(* CODESYS project Tc3_Mc3PlanarMotion.library
   TcLibraryId: Beckhoff Automation GmbH|Tc3_Mc3PlanarMotion|3.4.67.0
   Company: Beckhoff Automation GmbH
   DefaultNamespace: Tc3_Mc3PlanarMotion
   Version: 3.4.67.0
   Placeholder: Tc3_Mc3PlanarMotion
   Title: Tc3_Mc3PlanarMotion

Project tree, tasks and I/O mapping:
  libraries: Tc3_Physics, 3.4.67.0 (Beckhoff Automation GmbH)
  Version/
    global variables Global_Version
  POUs/
    function block MC_PlanarEnvironment [ST]: FB_init, FB_reinit, FB_exit, Clear, AddStator, CreateBoundary, Update, AddToGroup, RemoveFromGroup, GetPlanarObjectInfo
    function block MC_PlanarPart [ST]: FB_init, FB_reinit, FB_exit, Initialize, ActivatePosition, ForceEnable, AllowEnable, ForceDisable, Reset, GetPosition, IsInitialized, State, IsDisableForced, PositionIndex
    function block MC_PlanarGroup [ST]: FB_init, FB_reinit, FB_exit, Enable, Disable, Reset, Update
    function block MC_PlanarTrack [ST]: FB_init, FB_reinit, FB_exit, Clear, AppendPosition, AppendLine, AppendCircle, CloseLoop, StartFromTrack, EndAtTrack, StartFromTrackAdvanced, EndAtTrackAdvanced, Enable, Disable, Reset, GetArcLengthClosestTo, GetPositionAt, GetLength, GetPlanarObjectInfo, Update, AddToGroup, RemoveFromGroup
    function block MC_PlanarTrackTrail [ST]: FB_init, FB_reinit, FB_exit, Clear, AddTrack, GetTrackOidAt, TrackCount
    function block MC_PlanarMover [ST]: FB_init, FB_reinit, FB_exit, MoveToPosition, JoinTrack, LeaveTrack, MoveOnTrack, GearInPosOnTrack, GearInPosOnTrackWithMasterMover, MoveX, MoveY, MoveZ, MoveA, MoveB, MoveC, MoveRelativeX, MoveRelativeY, MoveRelativeC, MoveVelocityX, MoveVelocityY, MoveVelocityC, AdoptTrackOrientation, Halt, Enable, Disable, Reset, Update, SetPosition, StartExternalSetpointGeneration, StopExternalSetpointGeneration, SetExternalSetpoint, SetExternalSetpointReferenceId, RaiseError, AddToGroup, RemoveFromGroup, GetPositionOnCurrentPart, GetTrackTrailInformation, GetPlanarObjectInfo, MoverHardwareOid
    function block MC_PlanarFeedbackBase [ST]: FB_init, FB_reinit, FB_exit
    function block MC_PlanarFeedback [ST]: FB_init, FB_reinit, FB_exit, Update
    function block MC_PlanarFeedbackInSync [ST]: FB_init, FB_reinit, FB_exit
    function block MC_PlanarFeedbackGearInPosOnTrack [ST]: FB_init, FB_reinit, FB_exit, Update
    function block MC_PlanarFeedbackGearInPosOnTrackWithMasterMover [ST]: FB_init, FB_reinit, FB_exit, Update
  DUTs/
    Enums/
      data type MC_SET_POSITION_MODE
      data type MC_DIRECTION
      data type MC_SYNC_DIRECTIONS
      data type EPlanarObjectType
    Structs/
      data type PlanarObjectInfo
      data type ST_MoveToPositionOptions
      data type ST_JoinTrackOptions
      data type ST_LeaveTrackOptions
      data type ST_MoveOnTrackOptions
      data type ST_GearInPosOnTrackOptions
      data type ST_GearInPosOnTrackWithMasterMoverOptions
      data type ST_ExternalSetpointGenerationOptions
      data type ST_MoveCOptions
      data type ST_AdoptTrackOrientationOptions
      data type ST_StartFromTrackAdvancedOptions
      data type ST_EndAtTrackAdvancedOptions
    data type CDT_PLCTOMC_PLANAR_MOVER
    data type CDT_MCTOPLC_PLANAR_MOVER
*)

// DUTs/CDT_PLCTOMC_PLANAR_MOVER

(* Contains the information of the Planar Mover passed from PLC to MC. *)
	{attribute 'TcIecLibraryType'}
TYPE CDT_PLCTOMC_PLANAR_MOVER : 
	STRUCT
		(* Mover standard data that is transferred from this function block to the Planar Mover. *)
		{attribute 'TcPointerMapping'}
		 {attribute 'GUID' := 'BC77732B-A71D-4084-AA53-85A5016932F3'}
		 {attribute 'Namespace' := 'MC'}
		STD : REFERENCE TO CDT_PLCTOMC_PLANAR_MOVER_STD;
	END_STRUCT
END_TYPE

// DUTs/CDT_MCTOPLC_PLANAR_MOVER

(* Contains the information of the Planar Mover passed from MC to PLC. *)
	{attribute 'TcIecLibraryType'}
TYPE CDT_MCTOPLC_PLANAR_MOVER : 
	STRUCT
		(* Mover standard data that is transferred from the Planar Mover to this function block. *)
		{attribute 'TcPointerMapping'}
		 {attribute 'GUID' := '7D131116-81E4-45B0-AC50-A71EE4201E30'}
		 {attribute 'Namespace' := 'MC'}
		STD : REFERENCE TO CDT_MCTOPLC_PLANAR_MOVER_STD;
		(* Mover setpoint data that is transferred from the Planar Mover to this function block. *)
		{attribute 'TcPointerMapping'}
		 {attribute 'GUID' := 'D7D4F146-9962-4745-8631-17F5FB457164'}
		 {attribute 'Namespace' := 'MC'}
		SET : REFERENCE TO CDT_MCTOPLC_PLANAR_MOVER_SET;
		(* Mover actpoint data that is transferred from the Planar Mover to this function block. *)
		{attribute 'TcPointerMapping'}
		 {attribute 'GUID' := 'F18FBB92-D68F-43D8-95AE-0E42EDCD14E2'}
		 {attribute 'Namespace' := 'MC'}
		ACT : REFERENCE TO CDT_MCTOPLC_PLANAR_MOVER_ACT;
		(* Mover coordinate mode information that is transferred from the Planar Mover to this function block. *)
		{attribute 'TcPointerMapping'}
		 {attribute 'GUID' := 'B2D0D1AF-2BA9-49BA-AF3F-BC95009CD9CD'}
		 {attribute 'Namespace' := 'MC'}
		COORDMODE : REFERENCE TO CDT_MCTOPLC_PLANAR_MOVER_COORDMODE;
		(* Mover busy information that is transferred from the Planar Mover to this function block. *)
		{attribute 'TcPointerMapping'}
		 {attribute 'GUID' := 'DB4B14FF-1923-4ED2-A97C-3D3120BDBDAA'}
		 {attribute 'Namespace' := 'MC'}
		SETONTRACK : REFERENCE TO CDT_MCTOPLC_PLANAR_MOVER_TRACK;
	END_STRUCT
END_TYPE

// DUTs/Enums/MC_SET_POSITION_MODE

(* Indicates the external setpoint generation mode. *)
	{attribute 'TcIecLibraryType'}
{attribute 'BaseTypeGUID' := 'C4BA2B11-27FE-4956-B736-B8F79E7E1624'}
{attribute 'BaseTypeNamespace' := 'MC'}
{attribute 'qualified_only'}
{attribute 'strict'}
{attribute 'to_string'}
{attribute 'obsolete‘ :=‘Please use type MC_EXTERNAL_SET_POSITION_MODE instead'}
TYPE MC_SET_POSITION_MODE : MC_EXTERNAL_SET_POSITION_MODE;
END_TYPE

// DUTs/Enums/MC_DIRECTION

(* Indicates the movement direction of the Planar Mover on a Planar Track. *)
	{attribute 'TcIecLibraryType'}
{attribute 'qualified_only'}
{attribute 'to_string'}
TYPE MC_DIRECTION : (
	mcDirectionNonModulo:=0, 	(* The Planar Mover moves to the absolute value of the target position. Depending on the current position, this may induce forward or backward movement. On looped tracks, multiple passes are possible. *)
	mcDirectionPositive:=1, 	(* The Planar Mover moves to the target position in a forward direction. No backward movement is allowed. *)
	mcDirectionShortestWay:=2, 	(* The Planar Mover takes the shortest way to the target position. May induce forward or backward movement. *)
	mcDirectionNegative:=3	(* The Planar Mover moves to the target position in a backward direction. No forward movement is allowed. *)
) UINT;
END_TYPE

// DUTs/Enums/MC_SYNC_DIRECTIONS

(* Directions in which a slave is allowed to move during synchronizing phase. *)
	{attribute 'TcIecLibraryType'}
{attribute 'qualified_only'}
{attribute 'to_string'}
TYPE MC_SYNC_DIRECTIONS : (
		{attribute 'hide'}
Invalid:=0, 	(* Indicates invalid information, e.g. no connection or component not yet ready. *)
	Positive:=1, 	(* Movement is allowed only in positive direction while synchronizing. *)
	Negative:=2, 	(* Movement is allowed only in negative direction while synchronizing. *)
	Both:=3	(* Movement is allowed in any direction while synchronizing. *)
) UINT := Invalid;
END_TYPE

// DUTs/Enums/EPlanarObjectType

(* Identifies a planar object type. *)
	{attribute 'TcIecLibraryType'}
{attribute 'qualified_only'}
{attribute 'to_string'}
TYPE EPlanarObjectType : (
	Invalid:=0, 	(* Indicates invalid information, e.g. no connection or component not yet ready. *)
	None:=301, 	(* No planar object. *)
	Mover:=302, 	(* Planar Mover. *)
	Track:=303, 	(* Planar Track. *)
	Environment:=304	(* Planar Environment. *)
) UINT;
END_TYPE

// DUTs/Structs/PlanarObjectInfo

(* Identifies a planar object uniquely by object id and type. *)
	{attribute 'TcIecLibraryType'}
TYPE PlanarObjectInfo : 
	STRUCT
		(* Object type. *)
		 {attribute 'GUID' := '76890AE9-CB7E-444D-A716-1872FD85E0C0'}
		ObjectType : EPlanarObjectType;
		 {attribute 'hide'}
		_reserved1 : UINT;
		(* Object id. *)
		Id : UDINT;
	END_STRUCT
END_TYPE

// DUTs/Structs/ST_MoveToPositionOptions

(* Options for the "MoveToPosition" command of the Planar Mover. *)
	{attribute 'TcIecLibraryType'}
TYPE ST_MoveToPositionOptions : 
	STRUCT
		(* If true, the target orientation is also reached at the end of the movement. *)
		useOrientation : BOOL := TRUE;
	END_STRUCT
END_TYPE

// DUTs/Structs/ST_JoinTrackOptions

(* Options for the "JoinTrack" command of the Planar Mover. *)
	{attribute 'TcIecLibraryType'}
TYPE ST_JoinTrackOptions : 
	STRUCT
		(* If true, the target orientation is also reached at the end of the movement. *)
		useOrientation : BOOL := TRUE;
	END_STRUCT
END_TYPE

// DUTs/Structs/ST_LeaveTrackOptions

(* Options for the "LeaveTrack" command of the Planar Mover. *)
	{attribute 'TcIecLibraryType'}
TYPE ST_LeaveTrackOptions : 
	STRUCT
		(* If true, the target orientation is also reached at the end of the movement. *)
		useOrientation : BOOL := TRUE;
	END_STRUCT
END_TYPE

// DUTs/Structs/ST_MoveOnTrackOptions

(* Options for the "MoveOnTrack" command of the Planar Mover. *)
	{attribute 'TcIecLibraryType'}
TYPE ST_MoveOnTrackOptions : 
	STRUCT
		(* Minimal distance [mm] to next Planar Mover on track. *)
		gap : LREAL := 200.0;
		(* Direction in which the target is approached. *)
		 {attribute 'GUID' := 'FA9CA56B-5BDF-42DB-BC74-B14868EB8B42'}
		direction : MC_DIRECTION := MC_DIRECTION.mcDirectionNonModulo;
		 {attribute 'hide'}
		_reserved1 : UINT;
		(* Addition turns to move in modulo movement (positive or negative). *)
		additionalTurns : UDINT := 0;
		(* Tolerance "window" [mm] in modulo movement. *)
		moduloTolerance : LREAL := 0.0;
		(* The way in which dynamics are planned on track. *)
		 {attribute 'GUID' := '51EC8EBA-E260-4EDC-94C0-5ED02ABD2F9A'}
		 {attribute 'Namespace' := 'MC'}
		dynamicMode : MC_DYNAMICS_REDUCTION_MODE := MC_DYNAMICS_REDUCTION_MODE.None;
		(* The way in which gap control is done with all neighbors on track. *)
		 {attribute 'GUID' := '50FEC5F2-C9A2-49A2-AB32-4764BBA0A649'}
		 {attribute 'Namespace' := 'MC'}
		gapMode : MC_GAP_MODE_ON_TRACK := MC_GAP_MODE_ON_TRACK.Standard1D;
		 {attribute 'hide'}
		_reserved2 : UDINT;
	END_STRUCT
END_TYPE

// DUTs/Structs/ST_GearInPosOnTrackOptions

(* Options for the "GearInPosOnTrack" command of the Planar Mover. *)
	{attribute 'TcIecLibraryType'}
TYPE ST_GearInPosOnTrackOptions : 
	STRUCT
		(* Minimal distance [mm] to next Planar Mover on track. *)
		gap : LREAL := 200.0;
		(* Tolerance in absolute value [mm] of position difference to master axis for inSync flag. *)
		inSyncToleranceDistance : LREAL := 0.0;
		(* Direction in which the slave sync position is approached. Applies only to closed-loop tracks; use the default value for open tracks. *)
		 {attribute 'GUID' := 'FA9CA56B-5BDF-42DB-BC74-B14868EB8B42'}
		directionSlaveSyncPosition : MC_DIRECTION := MC_DIRECTION.mcDirectionNonModulo;
		 {attribute 'hide'}
		_reserved1 : UINT;
		(* Additional turns for slave sync position. Applies only to closed-loop tracks; use the default value for open tracks. *)
		{attribute 'hide'}
		additionalTurnsSlaveSyncPosition : UDINT := 0;
		(* Tolerance "window" [mm] for slave sync position. Applies only to closed-loop tracks; use the default value for open tracks. *)
		moduloToleranceSlaveSyncPosition : LREAL := 0.0;
		(* Directions in which the slave is allowed to move while in synchronizing phase. *)
		 {attribute 'GUID' := 'FB609C0C-2EEE-47C8-81DA-1811E3534906'}
		allowedSlaveSyncDirections : MC_SYNC_DIRECTIONS := MC_SYNC_DIRECTIONS.Positive;
		 {attribute 'hide'}
		_reserved2 : ARRAY [1..6] OF USINT;
	END_STRUCT
END_TYPE

// DUTs/Structs/ST_GearInPosOnTrackWithMasterMoverOptions

(* Options for the "GearInPosOnTrackWithMasterMover" command of the Planar Mover. *)
	{attribute 'TcIecLibraryType'}
TYPE ST_GearInPosOnTrackWithMasterMoverOptions : 
	STRUCT
		(* Minimal distance [mm] to next Planar Mover on track. *)
		gap : LREAL := 200.0;
		(* Tolerance in absolute value [mm] of position difference to master axis for inSync flag. *)
		inSyncToleranceDistance : LREAL := 0.0;
		(* Direction in which the slave sync position is approached. Applies only to closed-loop tracks; use the default value for open tracks. *)
		 {attribute 'GUID' := 'FA9CA56B-5BDF-42DB-BC74-B14868EB8B42'}
		directionSlaveSyncPosition : MC_DIRECTION := MC_DIRECTION.mcDirectionNonModulo;
		 {attribute 'hide'}
		_reserved1 : UINT;
		(* Additional turns for slave sync position. Applies only to closed-loop tracks; use the default value for open tracks. *)
		{attribute 'hide'}
		additionalTurnsSlaveSyncPosition : UDINT := 0;
		(* Tolerance "window" [mm] for slave sync position. Applies only to closed-loop tracks; use the default value for open tracks. *)
		moduloToleranceSlaveSyncPosition : LREAL := 0.0;
		(* Direction in which the master sync position is approached. Applies only to closed-loop tracks; use the default value for open tracks. *)
		 {attribute 'GUID' := 'FA9CA56B-5BDF-42DB-BC74-B14868EB8B42'}
		directionMasterSyncPosition : MC_DIRECTION := MC_DIRECTION.mcDirectionNonModulo;
		 {attribute 'hide'}
		_reserved2 : UINT;
		(* Additional turns for master sync position. Applies only to closed-loop tracks; use the default value for open tracks. *)
		{attribute 'hide'}
		additionalTurnsMasterSyncPosition : UDINT := 0;
		(* Tolerance "window" [mm] for master sync position. Applies only to closed-loop tracks; use the default value for open tracks. *)
		moduloToleranceMasterSyncPosition : LREAL := 0.0;
		(* Directions in which the slave is allowed to move while in synchronizing phase. *)
		 {attribute 'GUID' := 'FB609C0C-2EEE-47C8-81DA-1811E3534906'}
		allowedSlaveSyncDirections : MC_SYNC_DIRECTIONS := MC_SYNC_DIRECTIONS.Positive;
		(* If TRUE, the slave PlanarMover will proceed to follow the master PlanarMover after the latter has traversed the masterSyncPosition. In this case the PlanarTrackTrail describes the slave's path towards the masterSyncPosition. If FALSE, the slave moves exclusively on the PlanarTrackTrail specified. *)
		followMover : BOOL := FALSE;
		 {attribute 'hide'}
		_reserved3 : ARRAY [1..5] OF USINT;
	END_STRUCT
END_TYPE

// DUTs/Structs/ST_ExternalSetpointGenerationOptions

(* Options for the "ExternalSetpointGeneration" command of the Planar Mover. *)
	{attribute 'TcIecLibraryType'}
TYPE ST_ExternalSetpointGenerationOptions : 
	STRUCT
		(* Mode can be relative or absolute, relative can be used parallel to all other commands, absolute only alone. *)
		 {attribute 'GUID' := 'C4BA2B11-27FE-4956-B736-B8F79E7E1624'}
		 {attribute 'Namespace' := 'MC'}
		mode : MC_EXTERNAL_SET_POSITION_MODE := MC_EXTERNAL_SET_POSITION_MODE.Absolute;
	END_STRUCT
END_TYPE

// DUTs/Structs/ST_MoveCOptions

(* Options for the "MoveC" command of the Planar Mover. *)
	{attribute 'TcIecLibraryType'}
TYPE ST_MoveCOptions : 
	STRUCT
		(* Addition turns to move in modulo movement (positive or negative). *)
		additionalTurns : UDINT := 0;
		(* Direction in which the target is approached. *)
		 {attribute 'GUID' := 'FA9CA56B-5BDF-42DB-BC74-B14868EB8B42'}
		direction : MC_DIRECTION := MC_DIRECTION.mcDirectionNonModulo;
		 {attribute 'hide'}
		_reserved1 : UINT;
	END_STRUCT
END_TYPE

// DUTs/Structs/ST_AdoptTrackOrientationOptions

(* Options for the "AdoptTrackOrientation" command of the Planar Mover. *)
	{attribute 'TcIecLibraryType'}
TYPE ST_AdoptTrackOrientationOptions : 
	STRUCT
		(* Addition turns to move in modulo movement (positive or negative). *)
		additionalTurns : UDINT := 0;
		(* Direction in which the target is approached. *)
		 {attribute 'GUID' := 'FA9CA56B-5BDF-42DB-BC74-B14868EB8B42'}
		direction : MC_DIRECTION := MC_DIRECTION.mcDirectionShortestWay;
		 {attribute 'hide'}
		_reserved1 : UINT;
	END_STRUCT
END_TYPE

// DUTs/Structs/ST_StartFromTrackAdvancedOptions

(* Options for the "StartFromTrackAdvanced" command of the Planar Track. *)
	{attribute 'TcIecLibraryType'}
TYPE ST_StartFromTrackAdvancedOptions : 
	STRUCT
		(* The index of the position in which the part of this track is for track connection. *)
		thisTrackPartPositionIndex : UDINT := 0;
		(* The index of the position in which the part of the other track is for track connection. *)
		otherTrackPartPositionIndex : UDINT := 0;
		(* If FALSE, the tracks are connected not only in the given positions configuration of their parts but also in all other (geometrically compatible) locations, otherwise only the specified location is connected. *)
		linkOnlyInSpecifiedPartPositions : BOOL := FALSE;
		 {attribute 'hide'}
		_reserved1 : ARRAY [1..3] OF USINT;
	END_STRUCT
END_TYPE

// DUTs/Structs/ST_EndAtTrackAdvancedOptions

(* Options for the "EndAtTrackAdvanced" command of the Planar Track. *)
	{attribute 'TcIecLibraryType'}
TYPE ST_EndAtTrackAdvancedOptions : 
	STRUCT
		(* The index of the position in which the part of this track is for track connection. *)
		thisTrackPartPositionIndex : UDINT := 0;
		(* The index of the position in which the part of the other track is for track connection. *)
		otherTrackPartPositionIndex : UDINT := 0;
		(* If FALSE, the tracks are connected not only in the given positions configuration of their parts but also in all other (geometrically compatible) locations, otherwise only the specified location is connected. *)
		linkOnlyInSpecifiedPartPositions : BOOL := FALSE;
		 {attribute 'hide'}
		_reserved1 : ARRAY [1..3] OF USINT;
	END_STRUCT
END_TYPE

// Version/Global_Version
{attribute 'TcGenerated'}
// This function has been automatically generated from the project information.
VAR_GLOBAL CONSTANT
	{attribute 'const_non_replaced'}
	{attribute 'linkalways'}
	stLibVersion_Tc3_Mc3PlanarMotion : ST_LibVersion := (iMajor := 3, iMinor := 4, iBuild := 67, iRevision := 0, sVersion := '3.4.67.0');
	{attribute 'const_non_replaced'}
	{attribute 'linkalways'}
	sLibraryId_Tc3_Mc3PlanarMotion : String := 'Beckhoff Automation GmbH|Tc3_Mc3PlanarMotion|3.4.67.0';
END_VAR

// POUs/MC_PlanarEnvironment

	{attribute 'c++_compatible'}
	{attribute 'external_name' := 'MC_PlanarEnvironment_GUID_A74DE1F5_BE7B_A0CE_0F10_191560964433'}
	{attribute 'TcIecLibraryType'}
	{attribute 'no_explicit_call' :='do not call this POU directly'}
	{attribute 'no_assign_warning'}
	(* A Planar Environment object specifies the environment that Planar Movers can move in. It contains information about the stator objects and boundaries of the movement area. *)
	FUNCTION_BLOCK MC_PlanarEnvironment
	VAR
		 {attribute 'hide'}
		_reserved1 : ARRAY [1..4] OF UINT_8_16;
	END_VAR
	VAR_INPUT
		(* Environment data that is transferred from the Planar Environment to this function block. *)
		 {attribute 'GUID' := '79107B5F-AFEC-4E5A-AF95-460E7D782CE1'}
		 {attribute 'Namespace' := 'MC'}
		MCTOPLC_STD AT %I* : CDT_MCTOPLC_PLANAR_ENVIRONMENT;
	END_VAR
	VAR_OUTPUT
		(* Flag indicating a Planar Environment error. *)
		Error : BOOL;
	END_VAR
	VAR
		 {attribute 'hide'}
		_reserved2 : ARRAY [1..3] OF USINT;
	END_VAR
	VAR_OUTPUT
		(* Error id indicating the Planar Environment error type. *)
		ErrorId : UDINT;
	END_VAR
	VAR
		 {attribute 'hide'}
		_reserved3 : ARRAY [1..4] OF UINT_8_16;
	END_VAR


	(* Internal method *)
	{attribute 'hide'}
	METHOD FB_init : BOOL
	VAR_INPUT
		(*  if TRUE, the retain variables are initialized (warm start / cold start) *)
		bInitRetains : BOOL;
		(*  if TRUE, the instance afterwards gets moved into the copy code (online change) *)
		bInCopyCode : BOOL;
	END_VAR
END_METHOD


	(* Internal method *)
	{attribute 'hide'}
	METHOD FB_reinit : BOOL
END_METHOD


	(* Internal method *)
	{attribute 'hide'}
	METHOD FB_exit : BOOL
	VAR_INPUT
		(*  if TRUE, the exit method is called for exiting an instance that is copied afterwards (online change). *)
		bInCopyCode : BOOL;
	END_VAR
END_METHOD


	(* Clears the Planar Environment (stators and boundary). *)
	METHOD Clear
	VAR_INPUT
		(* The feedback object for the command. *)
 {attribute 'GUID' := '8FADE443-0B9B-A171-01FE-C51D234B86F7'}
				commandFeedback : REFERENCE TO MC_PlanarFeedback;
	END_VAR
END_METHOD


	(* Adds a stator to the Planar Environment. *)
	METHOD AddStator
	VAR_INPUT
		(* The feedback object for the command. *)
 {attribute 'GUID' := '8FADE443-0B9B-A171-01FE-C51D234B86F7'}
				commandFeedback : REFERENCE TO MC_PlanarFeedback;
		(* The lower x position [mm] of the stator. *)
		lowerX : LREAL;
		(* The lower y position [mm] of the stator. *)
		lowerY : LREAL;
	END_VAR
END_METHOD


	(* Creates a boundary for the Planar Environment based on the previously added stator information or hardware information. *)
	METHOD CreateBoundary
	VAR_INPUT
		(* The feedback object for the command. *)
 {attribute 'GUID' := '8FADE443-0B9B-A171-01FE-C51D234B86F7'}
				commandFeedback : REFERENCE TO MC_PlanarFeedback;
	END_VAR
END_METHOD


	(* Synchronizes the object state. Call once per PLC cycle. *)
	METHOD Update
END_METHOD


	(* Adds the Planar Environment to the given Planar Group. *)
	METHOD AddToGroup
	VAR_INPUT
		(* The feedback object for the command. *)
 {attribute 'GUID' := '8FADE443-0B9B-A171-01FE-C51D234B86F7'}
				commandFeedback : REFERENCE TO MC_PlanarFeedback;
	END_VAR
	VAR_IN_OUT
		(* The Planar Group that the mover joins. *)
 {attribute 'GUID' := '311812D6-6FBB-A2BC-1644-8B3C8413ECE6'}
				group : MC_PlanarGroup;
	END_VAR
END_METHOD


	(* Removes the Planar Environment from its current Planar Group, i.e. disables collision checks. *)
	METHOD RemoveFromGroup
	VAR_INPUT
		(* The feedback object for the command. *)
 {attribute 'GUID' := '8FADE443-0B9B-A171-01FE-C51D234B86F7'}
				commandFeedback : REFERENCE TO MC_PlanarFeedback;
	END_VAR
END_METHOD


	(* Returns environment object info (type: environment, id: OID of nc environment). *)
	METHOD GetPlanarObjectInfo : PlanarObjectInfo
END_METHOD

END_FUNCTION_BLOCK

// POUs/MC_PlanarFeedback

	{attribute 'c++_compatible'}
	{attribute 'external_name' := 'MC_PlanarFeedback_GUID_8FADE443_0B9B_A171_01FE_C51D234B86F7'}
	{attribute 'TcIecLibraryType'}
	{attribute 'no_assign_warning'}
	(* Displays specific command status information for an associated command, given back by the MC Project. *)
	FUNCTION_BLOCK MC_PlanarFeedback EXTENDS MC_PlanarFeedbackBase 
	VAR_OUTPUT
		(* Indicates the command is done, i.e. execution of the command finished successfully. *)
		Done : BOOL;
	END_VAR
	VAR
		 {attribute 'hide'}
		_reserved1_1 : UINT_24_56;
	END_VAR


	(* Internal method *)
	{attribute 'hide'}
	METHOD FB_init : BOOL
	VAR_INPUT
		(*  if TRUE, the retain variables are initialized (warm start / cold start) *)
		bInitRetains : BOOL;
		(*  if TRUE, the instance afterwards gets moved into the copy code (online change) *)
		bInCopyCode : BOOL;
	END_VAR
END_METHOD


	(* Internal method *)
	{attribute 'hide'}
	METHOD FB_reinit : BOOL
END_METHOD


	(* Internal method *)
	{attribute 'hide'}
	METHOD FB_exit : BOOL
	VAR_INPUT
		(*  if TRUE, the exit method is called for exiting an instance that is copied afterwards (online change). *)
		bInCopyCode : BOOL;
	END_VAR
END_METHOD


	(* Updates internal state of the object. *)
	METHOD Update
END_METHOD

END_FUNCTION_BLOCK

// POUs/MC_PlanarFeedbackBase

	{attribute 'c++_compatible'}
	{attribute 'external_name' := 'MC_PlanarFeedbackBase_GUID_8D287D70_7E86_A52F_2AC8_A8DD8A518824'}
	{attribute 'TcIecLibraryType'}
	{attribute 'no_explicit_call' :='do not call this POU directly'}
	{attribute 'no_assign_warning'}
	{attribute 'hide'}
	(* Displays general command status information for an associated command, given back by the MC Project. *)
	FUNCTION_BLOCK MC_PlanarFeedbackBase
	VAR
		 {attribute 'hide'}
		_reserved1 : UINT;
	END_VAR
	VAR_OUTPUT
		(* Indicates an active command, i.e. command was accepted and is being executed. *)
		Active : BOOL;
		(* Indicates a busy command, i.e. command is being processed, waiting for execution, or already executing (= also active). *)
		Busy : BOOL;
		(* Indicates the command is aborted, i.e. execution of the command finished due the start of other commands. *)
		Aborted : BOOL;
		(* Indicates the command has an error. *)
		Error : BOOL;
	END_VAR
	VAR
		 {attribute 'hide'}
		_reserved2 : UINT;
	END_VAR
	VAR_OUTPUT
		(* Indicates the error id of the command error. *)
		ErrorId : UDINT;
	END_VAR
	VAR
		 {attribute 'hide'}
		_reserved3 : UDINT;
	END_VAR
	VAR_OUTPUT
		(* Indicates which object one would collide with. *)
		 {attribute 'GUID' := '29463DBB-43C2-43AB-ADE2-B70446C51EDF'}
		objectInfo : PlanarObjectInfo;
	END_VAR
	VAR
		 {attribute 'hide'}
		_reserved4 : ARRAY [1..24] OF UINT_8_16;
	END_VAR


	(* Internal method *)
	{attribute 'hide'}
	METHOD FB_init : BOOL
	VAR_INPUT
		(*  if TRUE, the retain variables are initialized (warm start / cold start) *)
		bInitRetains : BOOL;
		(*  if TRUE, the instance afterwards gets moved into the copy code (online change) *)
		bInCopyCode : BOOL;
	END_VAR
END_METHOD


	(* Internal method *)
	{attribute 'hide'}
	METHOD FB_reinit : BOOL
END_METHOD


	(* Internal method *)
	{attribute 'hide'}
	METHOD FB_exit : BOOL
	VAR_INPUT
		(*  if TRUE, the exit method is called for exiting an instance that is copied afterwards (online change). *)
		bInCopyCode : BOOL;
	END_VAR
END_METHOD

END_FUNCTION_BLOCK

// POUs/MC_PlanarGroup

	{attribute 'c++_compatible'}
	{attribute 'external_name' := 'MC_PlanarGroup_GUID_311812D6_6FBB_A2BC_1644_8B3C8413ECE6'}
	{attribute 'TcIecLibraryType'}
	{attribute 'no_explicit_call' :='do not call this POU directly'}
	{attribute 'no_assign_warning'}
	(* A Planar Group object. Planar Movers and other objects added to the group perform collision checks against each other. *)
	FUNCTION_BLOCK MC_PlanarGroup
	VAR
		 {attribute 'hide'}
		_reserved1 : ARRAY [1..16] OF UINT_8_16;
	END_VAR
	VAR_INPUT
		(* Group data that is transferred from the Planar Group to this function block. *)
		 {attribute 'GUID' := 'E06D295F-3D94-4B18-B587-C89D73DA41F4'}
		 {attribute 'Namespace' := 'MC'}
		MCTOPLC_STD AT %I* : CDT_MCTOPLC_GROUP_PLANAR;
	END_VAR
	VAR_OUTPUT
		(* Flag indicating a Planar Group error. *)
		Error : BOOL;
	END_VAR
	VAR
		 {attribute 'hide'}
		_reserved2 : ARRAY [1..3] OF USINT;
	END_VAR
	VAR_OUTPUT
		(* Error id indicating the Planar Group error type. *)
		ErrorId : UDINT;
	END_VAR
	VAR
		 {attribute 'hide'}
		_reserved3 : UINT_0_32;
		 {attribute 'hide'}
		_reserved4 : ARRAY [1..4] OF UINT_8_16;
	END_VAR


	(* Internal method *)
	{attribute 'hide'}
	METHOD FB_init : BOOL
	VAR_INPUT
		(*  if TRUE, the retain variables are initialized (warm start / cold start) *)
		bInitRetains : BOOL;
		(*  if TRUE, the instance afterwards gets moved into the copy code (online change) *)
		bInCopyCode : BOOL;
	END_VAR
END_METHOD


	(* Internal method *)
	{attribute 'hide'}
	METHOD FB_reinit : BOOL
END_METHOD


	(* Internal method *)
	{attribute 'hide'}
	METHOD FB_exit : BOOL
	VAR_INPUT
		(*  if TRUE, the exit method is called for exiting an instance that is copied afterwards (online change). *)
		bInCopyCode : BOOL;
	END_VAR
END_METHOD


	(* Starts enabling the Planar Group. *)
	METHOD Enable
	VAR_INPUT
		(* The feedback object for the command. *)
 {attribute 'GUID' := '8FADE443-0B9B-A171-01FE-C51D234B86F7'}
				commandFeedback : REFERENCE TO MC_PlanarFeedback;
	END_VAR
END_METHOD


	(* Starts disabling the Planar Group. *)
	METHOD Disable
	VAR_INPUT
		(* The feedback object for the command. *)
 {attribute 'GUID' := '8FADE443-0B9B-A171-01FE-C51D234B86F7'}
				commandFeedback : REFERENCE TO MC_PlanarFeedback;
	END_VAR
END_METHOD


	(* Starts resetting the Planar Group. *)
	METHOD Reset
	VAR_INPUT
		(* The feedback object for the command. *)
 {attribute 'GUID' := '8FADE443-0B9B-A171-01FE-C51D234B86F7'}
				commandFeedback : REFERENCE TO MC_PlanarFeedback;
	END_VAR
END_METHOD


	(* Synchronizes the object state. Call once per PLC cycle. *)
	METHOD Update
END_METHOD

END_FUNCTION_BLOCK

// POUs/MC_PlanarPart

	{attribute 'c++_compatible'}
	{attribute 'external_name' := 'MC_PlanarPart_GUID_F385DE78_65E9_A0CB_0E07_650539B8B35D'}
	{attribute 'TcIecLibraryType'}
	{attribute 'no_explicit_call' :='do not call this POU directly'}
	{attribute 'no_assign_warning'}
	(* A Planar Part object represents the area that Planar Movers can move on. It contains information about the stator objects. *)
	FUNCTION_BLOCK MC_PlanarPart
	VAR_OUTPUT
		(* OID of the Planar Part. *)
		 {attribute 'GUID' := '18071995-0000-0000-0000-00000000000F'}
		PartOID : OTCID;
		(* Flag indicating a Planar Part error. *)
		Error : BOOL;
	END_VAR
	VAR
		 {attribute 'hide'}
		_reserved1 : ARRAY [1..3] OF USINT;
	END_VAR
	VAR_OUTPUT
		(* Error id indicating the Planar Part error type. *)
		ErrorId : UDINT;
	END_VAR
	VAR
		 {attribute 'hide'}
		_reserved2 : UINT_0_32;
		 {attribute 'hide'}
		_reserved3 : ARRAY [1..4] OF UINT_8_16;
		 {attribute 'hide'}
		_reserved4 : ARRAY [1..8] OF USINT;
	END_VAR


	(* Internal method *)
	{attribute 'hide'}
	METHOD FB_init : BOOL
	VAR_INPUT
		(*  if TRUE, the retain variables are initialized (warm start / cold start) *)
		bInitRetains : BOOL;
		(*  if TRUE, the instance afterwards gets moved into the copy code (online change) *)
		bInCopyCode : BOOL;
	END_VAR
END_METHOD


	(* Internal method *)
	{attribute 'hide'}
	METHOD FB_reinit : BOOL
END_METHOD


	(* Internal method *)
	{attribute 'hide'}
	METHOD FB_exit : BOOL
	VAR_INPUT
		(*  if TRUE, the exit method is called for exiting an instance that is copied afterwards (online change). *)
		bInCopyCode : BOOL;
	END_VAR
END_METHOD


	(* Initialize the Planar Part, i.e. connecting it to the MC via its OID. *)
	METHOD Initialize
	VAR_INPUT
		(* The feedback object for the command. *)
 {attribute 'GUID' := '8FADE443-0B9B-A171-01FE-C51D234B86F7'}
				commandFeedback : REFERENCE TO MC_PlanarFeedback;
		(* OID of the part. *)
 {attribute 'GUID' := '18071995-0000-0000-0000-00000000000F'}
				partOID : OTCID;
	END_VAR
	VAR_IN_OUT
		(* Environment the part is in. *)
 {attribute 'GUID' := 'A74DE1F5-BE7B-A0CE-0F10-191560964433'}
				environment : MC_PlanarEnvironment;
	END_VAR
END_METHOD


	(* Activates the position given by part position index. *)
	METHOD ActivatePosition
	VAR_INPUT
		(* The feedback object for the command. *)
 {attribute 'GUID' := '8FADE443-0B9B-A171-01FE-C51D234B86F7'}
				commandFeedback : REFERENCE TO MC_PlanarFeedback;
		(* Index of the position. *)
		positionIndex : UDINT;
	END_VAR
END_METHOD


	(* Removes force disable and enables the part. *)
	METHOD ForceEnable
	VAR_INPUT
		(* The feedback object for the command. *)
 {attribute 'GUID' := '8FADE443-0B9B-A171-01FE-C51D234B86F7'}
				commandFeedback : REFERENCE TO MC_PlanarFeedback;
	END_VAR
END_METHOD


	(* From now on the part can be enabled until ForceDisablePart is called. *)
	METHOD AllowEnable
	VAR_INPUT
		(* The feedback object for the command. *)
 {attribute 'GUID' := '8FADE443-0B9B-A171-01FE-C51D234B86F7'}
				commandFeedback : REFERENCE TO MC_PlanarFeedback;
	END_VAR
END_METHOD


	(* Disables the part and keeps it disabled until AllowEnabledPart is called. *)
	METHOD ForceDisable
	VAR_INPUT
		(* The feedback object for the command. *)
 {attribute 'GUID' := '8FADE443-0B9B-A171-01FE-C51D234B86F7'}
				commandFeedback : REFERENCE TO MC_PlanarFeedback;
	END_VAR
END_METHOD


	(* Resets the part. *)
	METHOD Reset
	VAR_INPUT
		(* The feedback object for the command. *)
 {attribute 'GUID' := '8FADE443-0B9B-A171-01FE-C51D234B86F7'}
				commandFeedback : REFERENCE TO MC_PlanarFeedback;
	END_VAR
END_METHOD


	(* Sets the values of the given position to the parts position values. *)
	METHOD GetPosition
	VAR_IN_OUT
		(* The position of the Planar Part. *)
 {attribute 'GUID' := '12927DD4-F3D1-1B21-A804-08BCF50529B3'}
		 {attribute 'Namespace' := 'Tc3_Physics'}
				position : PositionXYC;
	END_VAR
END_METHOD


{attribute 'monitoring' := 'call'}
	PROPERTY IsInitialized : BOOL
GET
END_GET
END_PROPERTY


{attribute 'monitoring' := 'call'}
	PROPERTY State : MC_PLANAR_STATE
GET
END_GET
END_PROPERTY


{attribute 'monitoring' := 'call'}
	PROPERTY IsDisableForced : BOOL
GET
END_GET
END_PROPERTY


{attribute 'monitoring' := 'call'}
	PROPERTY PositionIndex : UDINT
GET
END_GET
END_PROPERTY

END_FUNCTION_BLOCK

// POUs/MC_PlanarTrack

	{attribute 'c++_compatible'}
	{attribute 'external_name' := 'MC_PlanarTrack_GUID_9C7BCBA9_D9AF_AB6D_35ED_C2F4B777D1EA'}
	{attribute 'TcIecLibraryType'}
	{attribute 'no_explicit_call' :='do not call this POU directly'}
	{attribute 'no_assign_warning'}
	(* A track within a plane which Planar Movers can follow. Planar Movers on the track automatically avoid collisions with each other. The Planar Track can consist of several consecutive segments and be joined with other Planar Tracks at its start/end. *)
	FUNCTION_BLOCK MC_PlanarTrack
	VAR
		 {attribute 'hide'}
		_reserved1 : ARRAY [1..16] OF UINT_8_16;
	END_VAR
	VAR_INPUT
		(* Track data that is transferred from the Planar Track to this function block. *)
		 {attribute 'GUID' := '5769ADF0-D6E6-40D9-B474-790A2A7F1D1F'}
		 {attribute 'Namespace' := 'MC'}
		MCTOPLC_STD AT %I* : CDT_MCTOPLC_PLANAR_TRACK;
	END_VAR
	VAR_OUTPUT
		(* Flag indicating a Planar Track error. *)
		Error : BOOL;
	END_VAR
	VAR
		 {attribute 'hide'}
		_reserved2 : ARRAY [1..3] OF USINT;
	END_VAR
	VAR_OUTPUT
		(* Error id indicating the Planar Track error type. *)
		ErrorId : UDINT;
	END_VAR
	VAR
		 {attribute 'hide'}
		_reserved3 : UINT_0_32;
		 {attribute 'hide'}
		_reserved4 : ARRAY [1..4] OF UINT_8_16;
	END_VAR


	(* Internal method *)
	{attribute 'hide'}
	METHOD FB_init : BOOL
	VAR_INPUT
		(*  if TRUE, the retain variables are initialized (warm start / cold start) *)
		bInitRetains : BOOL;
		(*  if TRUE, the instance afterwards gets moved into the copy code (online change) *)
		bInCopyCode : BOOL;
	END_VAR
END_METHOD


	(* Internal method *)
	{attribute 'hide'}
	METHOD FB_reinit : BOOL
END_METHOD


	(* Internal method *)
	{attribute 'hide'}
	METHOD FB_exit : BOOL
	VAR_INPUT
		(*  if TRUE, the exit method is called for exiting an instance that is copied afterwards (online change). *)
		bInCopyCode : BOOL;
	END_VAR
END_METHOD


	(* Clears the geometric information of the Planar Track. *)
	METHOD Clear
	VAR_INPUT
		(* The feedback object for the command. *)
 {attribute 'GUID' := '8FADE443-0B9B-A171-01FE-C51D234B86F7'}
				commandFeedback : REFERENCE TO MC_PlanarFeedback;
	END_VAR
END_METHOD


	(* Appends a position to the Planar Track. *)
	METHOD AppendPosition
	VAR_INPUT
		(* The feedback object for the command. *)
 {attribute 'GUID' := '8FADE443-0B9B-A171-01FE-C51D234B86F7'}
				commandFeedback : REFERENCE TO MC_PlanarFeedback;
	END_VAR
	VAR_IN_OUT
		(* Position that is the new endpoint of the Planar Track. *)
 {attribute 'GUID' := '12927DD4-F3D1-1B21-A804-08BCF50529B3'}
		 {attribute 'Namespace' := 'Tc3_Physics'}
				position : PositionXYC;
	END_VAR
END_METHOD


	(* Appends a line to the Planar Track. *)
	METHOD AppendLine
	VAR_INPUT
		(* The feedback object for the command. *)
 {attribute 'GUID' := '8FADE443-0B9B-A171-01FE-C51D234B86F7'}
				commandFeedback : REFERENCE TO MC_PlanarFeedback;
	END_VAR
	VAR_IN_OUT
		(* Start position of the line. *)
 {attribute 'GUID' := '12927DD4-F3D1-1B21-A804-08BCF50529B3'}
		 {attribute 'Namespace' := 'Tc3_Physics'}
				start : PositionXYC;
		(* End position of the line, this position is the new endpoint of the Planar Track. *)
 {attribute 'GUID' := '12927DD4-F3D1-1B21-A804-08BCF50529B3'}
		 {attribute 'Namespace' := 'Tc3_Physics'}
				end : PositionXYC;
	END_VAR
END_METHOD


	(* Appends a circular arc to the Planar Track. *)
	METHOD AppendCircle
	VAR_INPUT
		(* The feedback object for the command. *)
 {attribute 'GUID' := '8FADE443-0B9B-A171-01FE-C51D234B86F7'}
				commandFeedback : REFERENCE TO MC_PlanarFeedback;
	END_VAR
	VAR_IN_OUT
		(* Start position of the circular arc. *)
 {attribute 'GUID' := '12927DD4-F3D1-1B21-A804-08BCF50529B3'}
		 {attribute 'Namespace' := 'Tc3_Physics'}
				start : PositionXYC;
		(* End position of the circular arc, this position is the new endpoint of the Planar Track. *)
 {attribute 'GUID' := '12927DD4-F3D1-1B21-A804-08BCF50529B3'}
		 {attribute 'Namespace' := 'Tc3_Physics'}
				end : PositionXYC;
		(* Center of the circular arc. *)
 {attribute 'GUID' := '97A8C469-9E33-1367-BD2B-4B487B94CC01'}
		 {attribute 'Namespace' := 'Tc3_Physics'}
				center : PositionXY;
	END_VAR
	VAR_INPUT
		(* Indicates if the clockwise circle is appended. *)
		clockwise : BOOL;
	END_VAR
END_METHOD


	(* Closes the loop of the Planar Track, no further part can be appended. *)
	METHOD CloseLoop
	VAR_INPUT
		(* The feedback object for the command. *)
 {attribute 'GUID' := '8FADE443-0B9B-A171-01FE-C51D234B86F7'}
				commandFeedback : REFERENCE TO MC_PlanarFeedback;
	END_VAR
END_METHOD


	(* Sets the other Planar Track's endpoint as start point of this Planar Track, transition is smooth. The other Planar Track is blocked for further changes (until it is cleared). *)
	METHOD StartFromTrack
	VAR_INPUT
		(* The feedback object for the command. *)
 {attribute 'GUID' := '8FADE443-0B9B-A171-01FE-C51D234B86F7'}
				commandFeedback : REFERENCE TO MC_PlanarFeedback;
	END_VAR
	VAR_IN_OUT
		(* The other Planar Track. *)
 {attribute 'GUID' := '9C7BCBA9-D9AF-AB6D-35ED-C2F4B777D1EA'}
				track : MC_PlanarTrack;
	END_VAR
END_METHOD


	(* Appends a smooth transition from the end of this Planar Track to the other Planar Track's start point. The Planar Track is blocked for further changes (until it is cleared). *)
	METHOD EndAtTrack
	VAR_INPUT
		(* The feedback object for the command. *)
 {attribute 'GUID' := '8FADE443-0B9B-A171-01FE-C51D234B86F7'}
				commandFeedback : REFERENCE TO MC_PlanarFeedback;
	END_VAR
	VAR_IN_OUT
		(* The other Planar Track. *)
 {attribute 'GUID' := '9C7BCBA9-D9AF-AB6D-35ED-C2F4B777D1EA'}
				track : MC_PlanarTrack;
	END_VAR
END_METHOD


	(* Sets the other Planar Track's endpoint as start point of this Planar Track, transition is smooth. The other Planar Track is blocked for further geometrical changes (until it is cleared). *)
	METHOD StartFromTrackAdvanced
	VAR_INPUT
		(* The feedback object for the command. *)
 {attribute 'GUID' := '8FADE443-0B9B-A171-01FE-C51D234B86F7'}
				commandFeedback : REFERENCE TO MC_PlanarFeedback;
	END_VAR
	VAR_IN_OUT
		(* The other Planar Track. *)
 {attribute 'GUID' := '9C7BCBA9-D9AF-AB6D-35ED-C2F4B777D1EA'}
				track : MC_PlanarTrack;
	END_VAR
	VAR_INPUT
		(* Options for the connection, i.e. which connections are closed. *)
 {attribute 'GUID' := 'BFAEC56B-EA59-4E6C-80D6-CFD454740FA4'}
				options : REFERENCE TO ST_StartFromTrackAdvancedOptions;
	END_VAR
END_METHOD


	(* Appends a smooth transition from the end of this Planar Track to the other Planar Track's start point. The Planar Track is blocked for further geometrical changes (until it is cleared). *)
	METHOD EndAtTrackAdvanced
	VAR_INPUT
		(* The feedback object for the command. *)
 {attribute 'GUID' := '8FADE443-0B9B-A171-01FE-C51D234B86F7'}
				commandFeedback : REFERENCE TO MC_PlanarFeedback;
	END_VAR
	VAR_IN_OUT
		(* The other Planar Track. *)
 {attribute 'GUID' := '9C7BCBA9-D9AF-AB6D-35ED-C2F4B777D1EA'}
				track : MC_PlanarTrack;
	END_VAR
	VAR_INPUT
		(* Options for the connection, i.e. which connections are closed. *)
 {attribute 'GUID' := 'BF8474CD-E31A-4854-97DD-B0AB77EF6586'}
				options : REFERENCE TO ST_EndAtTrackAdvancedOptions;
	END_VAR
END_METHOD


	(* Starts enabling the Planar Track. *)
	METHOD Enable
	VAR_INPUT
		(* The feedback object for the command. *)
 {attribute 'GUID' := '8FADE443-0B9B-A171-01FE-C51D234B86F7'}
				commandFeedback : REFERENCE TO MC_PlanarFeedback;
	END_VAR
END_METHOD


	(* Starts disabling the Planar Track. *)
	METHOD Disable
	VAR_INPUT
		(* The feedback object for the command. *)
 {attribute 'GUID' := '8FADE443-0B9B-A171-01FE-C51D234B86F7'}
				commandFeedback : REFERENCE TO MC_PlanarFeedback;
	END_VAR
END_METHOD


	(* Starts resetting the Planar Track. *)
	METHOD Reset
	VAR_INPUT
		(* The feedback object for the command. *)
 {attribute 'GUID' := '8FADE443-0B9B-A171-01FE-C51D234B86F7'}
				commandFeedback : REFERENCE TO MC_PlanarFeedback;
	END_VAR
END_METHOD


	(* Calculate the arc length value [mm] where the Planar Track is closest to a geometry's center point. *)
	METHOD GetArcLengthClosestTo : LREAL
	VAR_IN_OUT
		(* The geometry to check the arc length for. *)
 {attribute 'GUID' := '432B7521-EF05-1C03-897A-3B970F77C0D6'}
		 {attribute 'Namespace' := 'Tc3_Physics'}
				geometry : IPlcGeometry2D;
	END_VAR
END_METHOD


	(* Get a position on the Planar Track at a specific arc length value. *)
	METHOD GetPositionAt
	VAR_INPUT
		(* Arc length value where the position is evaluated. *)
		arcLength : LREAL;
	END_VAR
	VAR_IN_OUT
		(* The position at the specified arc parameter. *)
 {attribute 'GUID' := '12927DD4-F3D1-1B21-A804-08BCF50529B3'}
		 {attribute 'Namespace' := 'Tc3_Physics'}
				position : PositionXYC;
	END_VAR
END_METHOD


	(* Returns the Planar Track's length [mm], -1 return value indicates no connection to Nc Track. *)
	METHOD GetLength : LREAL
END_METHOD


	(* Returns track object info (type: track, id: OID of nc track). *)
	METHOD GetPlanarObjectInfo : PlanarObjectInfo
END_METHOD


	(* Synchronizes the object state. Call once per PLC cycle. *)
	METHOD Update
END_METHOD


	(* Adds the Planar Track to the given Planar Group. *)
	METHOD AddToGroup
	VAR_INPUT
		(* The feedback object for the command. *)
 {attribute 'GUID' := '8FADE443-0B9B-A171-01FE-C51D234B86F7'}
				commandFeedback : REFERENCE TO MC_PlanarFeedback;
	END_VAR
	VAR_IN_OUT
		(* The Planar Group that the mover joins. *)
 {attribute 'GUID' := '311812D6-6FBB-A2BC-1644-8B3C8413ECE6'}
				group : MC_PlanarGroup;
	END_VAR
END_METHOD


	(* Removes the Planar Track from its current Planar Group, i.e. disables collision checks. *)
	METHOD RemoveFromGroup
	VAR_INPUT
		(* The feedback object for the command. *)
 {attribute 'GUID' := '8FADE443-0B9B-A171-01FE-C51D234B86F7'}
				commandFeedback : REFERENCE TO MC_PlanarFeedback;
	END_VAR
END_METHOD

END_FUNCTION_BLOCK

// POUs/MC_PlanarTrackTrail

	{attribute 'c++_compatible'}
	{attribute 'external_name' := 'MC_PlanarTrackTrail_GUID_F8359FE7_9712_A2F1_01A5_A9544A0C00B7'}
	{attribute 'TcIecLibraryType'}
	{attribute 'no_explicit_call' :='do not call this POU directly'}
	{attribute 'no_assign_warning'}
	(* A list of distinct tracks each starting at the ending vertex of its predecessor. *)
	FUNCTION_BLOCK MC_PlanarTrackTrail
	VAR_OUTPUT
		(* Flag indicating a TrackTrail error. *)
		Error : BOOL;
	END_VAR
	VAR
		 {attribute 'hide'}
		_reserved1 : ARRAY [1..3] OF USINT;
	END_VAR
	VAR_OUTPUT
		(* Error id indicating the TrackTrail error type. *)
		ErrorId : UDINT;
		(* Number of tracks stored in this trail. *)
		{attribute 'hide'}
		Size : UDINT;
	END_VAR
	VAR
		 {attribute 'hide'}
		_reserved2 : UINT_0_32;
		 {attribute 'hide'}
		_reserved3 : ARRAY [1..20] OF UINT_8_16;
	END_VAR


	(* Internal method *)
	{attribute 'hide'}
	METHOD FB_init : BOOL
	VAR_INPUT
		(*  if TRUE, the retain variables are initialized (warm start / cold start) *)
		bInitRetains : BOOL;
		(*  if TRUE, the instance afterwards gets moved into the copy code (online change) *)
		bInCopyCode : BOOL;
	END_VAR
END_METHOD


	(* Internal method *)
	{attribute 'hide'}
	METHOD FB_reinit : BOOL
END_METHOD


	(* Internal method *)
	{attribute 'hide'}
	METHOD FB_exit : BOOL
	VAR_INPUT
		(*  if TRUE, the exit method is called for exiting an instance that is copied afterwards (online change). *)
		bInCopyCode : BOOL;
	END_VAR
END_METHOD


	(* Clears the TrackTrail. *)
	METHOD Clear
END_METHOD


	(* Adds a track to the TrackTrail. The track should start at the end vertex of the currently last track. *)
	METHOD AddTrack
	VAR_IN_OUT
		(* The track to be added to the end of the TrackTrail. *)
 {attribute 'GUID' := '9C7BCBA9-D9AF-AB6D-35ED-C2F4B777D1EA'}
				track : MC_PlanarTrack;
	END_VAR
END_METHOD


	(* Returns the oid of the track at the specified index [1, ..., size] in the trail. Zero is returned on error. *)
	METHOD GetTrackOidAt : OTCID
	VAR_INPUT
		(* Index of the track in the trail [1, ..., size]. *)
		index : UDINT;
	END_VAR
END_METHOD


{attribute 'monitoring' := 'call'}
	PROPERTY TrackCount : UDINT
GET
END_GET
END_PROPERTY

END_FUNCTION_BLOCK

// POUs/MC_PlanarMover

	{attribute 'c++_compatible'}
	{attribute 'external_name' := 'MC_PlanarMover_GUID_5D145DEA_6FDD_A2B2_3626_4BBE11F87E8C'}
	{attribute 'TcIecLibraryType'}
	{attribute 'no_explicit_call' :='do not call this POU directly'}
	{attribute 'no_assign_warning'}
	(* A Planar Mover object capable of moving within a plane. Limited movement vertical to the plane is available. *)
	FUNCTION_BLOCK MC_PlanarMover
	VAR_INPUT
		(* Mover data that is transferred from this function block to the Planar Mover. *)
		 {attribute 'GUID' := '0FD45376-89CE-4D41-87B5-C009E54908A1'}
		PLCTOMC AT %Q* : CDT_PLCTOMC_PLANAR_MOVER;
		(* Mover data that is transferred from the Planar Mover to this function block. *)
		 {attribute 'GUID' := 'EA1F10AA-0C64-4FA5-978B-F78C44393D9A'}
		MCTOPLC AT %I* : CDT_MCTOPLC_PLANAR_MOVER;
	END_VAR
	VAR
		 {attribute 'hide'}
		_reserved1 : ARRAY [1..32] OF UINT_8_16;
	END_VAR
	VAR_OUTPUT
		(* Flag indicating a Planar Mover error. *)
		Error : BOOL;
	END_VAR
	VAR
		 {attribute 'hide'}
		_reserved2 : ARRAY [1..3] OF USINT;
	END_VAR
	VAR_OUTPUT
		(* Error id indicating the Planar Mover error type. *)
		ErrorId : UDINT;
	END_VAR
	VAR
		 {attribute 'hide'}
		_reserved3 : ARRAY [1..4] OF UINT_8_16;
	END_VAR


	(* Internal method *)
	{attribute 'hide'}
	METHOD FB_init : BOOL
	VAR_INPUT
		(*  if TRUE, the retain variables are initialized (warm start / cold start) *)
		bInitRetains : BOOL;
		(*  if TRUE, the instance afterwards gets moved into the copy code (online change) *)
		bInCopyCode : BOOL;
	END_VAR
END_METHOD


	(* Internal method *)
	{attribute 'hide'}
	METHOD FB_reinit : BOOL
END_METHOD


	(* Internal method *)
	{attribute 'hide'}
	METHOD FB_exit : BOOL
	VAR_INPUT
		(*  if TRUE, the exit method is called for exiting an instance that is copied afterwards (online change). *)
		bInCopyCode : BOOL;
	END_VAR
END_METHOD


	(* Initiates a direct movement to the specified position. *)
	METHOD MoveToPosition
	VAR_INPUT
		(* The feedback object for the command. *)
 {attribute 'GUID' := '8FADE443-0B9B-A171-01FE-C51D234B86F7'}
				commandFeedback : REFERENCE TO MC_PlanarFeedback;
	END_VAR
	VAR_IN_OUT
		(* Target position for the movement. *)
 {attribute 'GUID' := '12927DD4-F3D1-1B21-A804-08BCF50529B3'}
		 {attribute 'Namespace' := 'Tc3_Physics'}
				targetPosition : PositionXYC;
	END_VAR
	VAR_INPUT
		(* Dynamic constraints for this movement. *)
 {attribute 'GUID' := '6C0A73A2-C983-14C5-9BC7-15048F604248'}
		 {attribute 'Namespace' := 'Tc3_Physics'}
				constraint : REFERENCE TO IPlcDynamicConstraint;
		(* Options for the movement. *)
 {attribute 'GUID' := '370F6D14-8A00-4DA3-B28C-5E648E8318EE'}
				options : REFERENCE TO ST_MoveToPositionOptions;
	END_VAR
END_METHOD


	(* Initiates a direct movement to the specified track. At the end of the movement the mover joins the track. *)
	METHOD JoinTrack
	VAR_INPUT
		(* The feedback object for the command. *)
 {attribute 'GUID' := '8FADE443-0B9B-A171-01FE-C51D234B86F7'}
				commandFeedback : REFERENCE TO MC_PlanarFeedback;
	END_VAR
	VAR_IN_OUT
		(* Target track for the movement. *)
 {attribute 'GUID' := '9C7BCBA9-D9AF-AB6D-35ED-C2F4B777D1EA'}
				targetTrack : MC_PlanarTrack;
	END_VAR
	VAR_INPUT
		(* Dynamic constraints for this movement. *)
 {attribute 'GUID' := '6C0A73A2-C983-14C5-9BC7-15048F604248'}
		 {attribute 'Namespace' := 'Tc3_Physics'}
				constraint : REFERENCE TO IPlcDynamicConstraint;
		(* Options for the movement. *)
 {attribute 'GUID' := '4F0F6069-E474-4F1D-AA55-745B4EFFC9D8'}
				options : REFERENCE TO ST_JoinTrackOptions;
	END_VAR
END_METHOD


	(* Initiates a direct movement to the specified position. At the beginning of the movement the track is left. *)
	METHOD LeaveTrack
	VAR_INPUT
		(* The feedback object for the command. *)
 {attribute 'GUID' := '8FADE443-0B9B-A171-01FE-C51D234B86F7'}
				commandFeedback : REFERENCE TO MC_PlanarFeedback;
	END_VAR
	VAR_IN_OUT
		(* Target position for the movement. *)
 {attribute 'GUID' := '12927DD4-F3D1-1B21-A804-08BCF50529B3'}
		 {attribute 'Namespace' := 'Tc3_Physics'}
				targetPosition : PositionXYC;
	END_VAR
	VAR_INPUT
		(* Dynamic constraints for this movement. *)
 {attribute 'GUID' := '6C0A73A2-C983-14C5-9BC7-15048F604248'}
		 {attribute 'Namespace' := 'Tc3_Physics'}
				constraint : REFERENCE TO IPlcDynamicConstraint;
		(* Options for the movement. *)
 {attribute 'GUID' := '143DAE7C-6701-4927-9629-961CD3D036A4'}
				options : REFERENCE TO ST_LeaveTrackOptions;
	END_VAR
END_METHOD


	(* Initiates a movement on the track to the specified position. *)
	METHOD MoveOnTrack
	VAR_INPUT
		(* The feedback object for the command. *)
 {attribute 'GUID' := '8FADE443-0B9B-A171-01FE-C51D234B86F7'}
				commandFeedback : REFERENCE TO MC_PlanarFeedback;
		(* Target track for the movement. If none is specified, this defaults to the current track. *)
 {attribute 'GUID' := '9C7BCBA9-D9AF-AB6D-35ED-C2F4B777D1EA'}
				targetTrack : REFERENCE TO MC_PlanarTrack;
		(* Target position [mm] on the target track. *)
		targetPositionOnTrack : LREAL;
		(* Constraint on maximal dynamics during the movement (V,A,D,J). *)
 {attribute 'GUID' := 'C03A5F50-C097-1CA1-90CF-4DB7CF7C4E51'}
		 {attribute 'Namespace' := 'Tc3_Physics'}
				constraint : REFERENCE TO DynamicConstraint_PathXY;
		(* Options for the movement. *)
 {attribute 'GUID' := '0B666056-872B-424E-B64A-F49609B0E127'}
				options : REFERENCE TO ST_MoveOnTrackOptions;
	END_VAR
END_METHOD


	(* Initiates a GearInPos movement along a specified trail. *)
	METHOD GearInPosOnTrack
	VAR_INPUT
		(* The command specific feedback object for the command. *)
 {attribute 'GUID' := '19C4A159-B3DC-ABFB-0783-72302E623B59'}
				commandFeedback : REFERENCE TO MC_PlanarFeedbackGearInPosOnTrack;
		(* Master axis being followed. *)
 {attribute 'GUID' := '18071995-0000-0000-0000-00000000000F'}
				masterAxis : OTCID;
		(* Track trail determining along which tracks the GearInPos movement is allowed to proceed. *)
 {attribute 'GUID' := 'F8359FE7-9712-A2F1-01A5-A9544A0C00B7'}
				trackTrail : REFERENCE TO MC_PlanarTrackTrail;
		(* Position of the master axis (interpreted as [mm]) at which the slave is inSync. *)
		masterSyncPosition : LREAL;
		(* Arc length [mm] on track given by slaveSyncPositionTrackOID at which the slave is inSync. Possibly interpreted in modulo fashion, depending on options. *)
		slaveSyncPosition : LREAL;
	END_VAR
	VAR_IN_OUT
		(* Track on which the slave is inSync. *)
 {attribute 'GUID' := '9C7BCBA9-D9AF-AB6D-35ED-C2F4B777D1EA'}
				slaveSyncPositionTrack : MC_PlanarTrack;
	END_VAR
	VAR_INPUT
		(* Constraint on maximal dynamics during the movement (V,A,D,J). *)
 {attribute 'GUID' := 'C03A5F50-C097-1CA1-90CF-4DB7CF7C4E51'}
		 {attribute 'Namespace' := 'Tc3_Physics'}
				constraint : REFERENCE TO DynamicConstraint_PathXY;
		(* Options for the movement. *)
 {attribute 'GUID' := 'A0DE3DE9-FE75-437E-9C4F-12CEF8F28D2C'}
				options : REFERENCE TO ST_GearInPosOnTrackOptions;
	END_VAR
END_METHOD


	(* Initiates a GearInPos movement along a specified trail, in which the master setpoints are provided by another PlanarMover. *)
	METHOD GearInPosOnTrackWithMasterMover
	VAR_INPUT
		(* The command specific feedback object for the command. *)
 {attribute 'GUID' := 'A3111726-B59C-A154-0494-25C5C4FF630E'}
				commandFeedback : REFERENCE TO MC_PlanarFeedbackGearInPosOnTrackWithMasterMover;
	END_VAR
	VAR_IN_OUT
		(* Master mover being followed. *)
 {attribute 'GUID' := '5D145DEA-6FDD-A2B2-3626-4BBE11F87E8C'}
				masterMover : MC_PlanarMover;
	END_VAR
	VAR_INPUT
		(* Track trail determining along which tracks the GearInPos movement is allowed to proceed. *)
 {attribute 'GUID' := 'F8359FE7-9712-A2F1-01A5-A9544A0C00B7'}
				trackTrail : REFERENCE TO MC_PlanarTrackTrail;
		(* Position of the master axis (interpreted as [mm]) at which the slave is inSync. *)
		masterSyncPosition : LREAL;
	END_VAR
	VAR_IN_OUT
		(* Track on which the master is inSync. *)
 {attribute 'GUID' := '9C7BCBA9-D9AF-AB6D-35ED-C2F4B777D1EA'}
				masterSyncPositionTrack : MC_PlanarTrack;
	END_VAR
	VAR_INPUT
		(* Arc length on track [mm] given by slaveSyncPositionTrackOID at which the slave is inSync. Possibly interpreted in modulo fashion, depending on options. *)
		slaveSyncPosition : LREAL;
	END_VAR
	VAR_IN_OUT
		(* Track on which the slave is inSync. *)
 {attribute 'GUID' := '9C7BCBA9-D9AF-AB6D-35ED-C2F4B777D1EA'}
				slaveSyncPositionTrack : MC_PlanarTrack;
	END_VAR
	VAR_INPUT
		(* Constraint on maximal dynamics during the movement (V,A,D,J). *)
 {attribute 'GUID' := 'C03A5F50-C097-1CA1-90CF-4DB7CF7C4E51'}
		 {attribute 'Namespace' := 'Tc3_Physics'}
				constraint : REFERENCE TO DynamicConstraint_PathXY;
		(* Options for the movement. *)
 {attribute 'GUID' := '5A8461CA-4052-4626-BC5D-1CE1B65683E0'}
				options : REFERENCE TO ST_GearInPosOnTrackWithMasterMoverOptions;
	END_VAR
END_METHOD


	(* Initiates a movement for the x component. *)
	METHOD MoveX
	VAR_INPUT
		(* The feedback object for the command. *)
 {attribute 'GUID' := '8FADE443-0B9B-A171-01FE-C51D234B86F7'}
				commandFeedback : REFERENCE TO MC_PlanarFeedback;
		(* Target position [mm] for the movement. *)
		targetPosition : LREAL;
		(* Reference system of the target position. *)
 {attribute 'GUID' := '18071995-0000-0000-0000-00000000000F'}
				refSys : OTCID;
		(* Dynamic constraints for this movement. *)
 {attribute 'GUID' := '6C0A73A2-C983-14C5-9BC7-15048F604248'}
		 {attribute 'Namespace' := 'Tc3_Physics'}
				constraint : REFERENCE TO IPlcDynamicConstraint;
	END_VAR
END_METHOD


	(* Initiates a movement for the y component. *)
	METHOD MoveY
	VAR_INPUT
		(* The feedback object for the command. *)
 {attribute 'GUID' := '8FADE443-0B9B-A171-01FE-C51D234B86F7'}
				commandFeedback : REFERENCE TO MC_PlanarFeedback;
		(* Target position [mm] for the movement. *)
		targetPosition : LREAL;
		(* Reference system of the target position. *)
 {attribute 'GUID' := '18071995-0000-0000-0000-00000000000F'}
				refSys : OTCID;
		(* Dynamic constraints for this movement. *)
 {attribute 'GUID' := '6C0A73A2-C983-14C5-9BC7-15048F604248'}
		 {attribute 'Namespace' := 'Tc3_Physics'}
				constraint : REFERENCE TO IPlcDynamicConstraint;
	END_VAR
END_METHOD


	(* Initiates a movement for the z component. *)
	METHOD MoveZ
	VAR_INPUT
		(* The feedback object for the command. *)
 {attribute 'GUID' := '8FADE443-0B9B-A171-01FE-C51D234B86F7'}
				commandFeedback : REFERENCE TO MC_PlanarFeedback;
		(* Target position [mm] for the movement. *)
		targetPosition : LREAL;
		(* Dynamic constraints for this movement. *)
 {attribute 'GUID' := '6C0A73A2-C983-14C5-9BC7-15048F604248'}
		 {attribute 'Namespace' := 'Tc3_Physics'}
				constraint : REFERENCE TO IPlcDynamicConstraint;
	END_VAR
END_METHOD


	(* Initiates a movement for the a component. *)
	METHOD MoveA
	VAR_INPUT
		(* The feedback object for the command. *)
 {attribute 'GUID' := '8FADE443-0B9B-A171-01FE-C51D234B86F7'}
				commandFeedback : REFERENCE TO MC_PlanarFeedback;
		(* Target position [deg] for the movement. *)
		targetPosition : LREAL;
		(* Dynamic constraints for this movement. *)
 {attribute 'GUID' := '6C0A73A2-C983-14C5-9BC7-15048F604248'}
		 {attribute 'Namespace' := 'Tc3_Physics'}
				constraint : REFERENCE TO IPlcDynamicConstraint;
	END_VAR
END_METHOD


	(* Initiates a movement for the b component. *)
	METHOD MoveB
	VAR_INPUT
		(* The feedback object for the command. *)
 {attribute 'GUID' := '8FADE443-0B9B-A171-01FE-C51D234B86F7'}
				commandFeedback : REFERENCE TO MC_PlanarFeedback;
		(* Target position [deg] for the movement. *)
		targetPosition : LREAL;
		(* Dynamic constraints for this movement. *)
 {attribute 'GUID' := '6C0A73A2-C983-14C5-9BC7-15048F604248'}
		 {attribute 'Namespace' := 'Tc3_Physics'}
				constraint : REFERENCE TO IPlcDynamicConstraint;
	END_VAR
END_METHOD


	(* Initiates a movement for the c component. *)
	METHOD MoveC
	VAR_INPUT
		(* The feedback object for the command. *)
 {attribute 'GUID' := '8FADE443-0B9B-A171-01FE-C51D234B86F7'}
				commandFeedback : REFERENCE TO MC_PlanarFeedback;
		(* Target position [deg] for the movement. *)
		targetPosition : LREAL;
		(* Dynamic constraints for this movement. *)
 {attribute 'GUID' := '6C0A73A2-C983-14C5-9BC7-15048F604248'}
		 {attribute 'Namespace' := 'Tc3_Physics'}
				constraint : REFERENCE TO IPlcDynamicConstraint;
		(* Options for the rotation. *)
 {attribute 'GUID' := '3968D894-10B1-4E26-AC44-4464598EF32A'}
				options : REFERENCE TO ST_MoveCOptions;
	END_VAR
END_METHOD


	(* Initiates a relative movement for the x component. *)
	METHOD MoveRelativeX
	VAR_INPUT
		(* The feedback object for the command. *)
 {attribute 'GUID' := '8FADE443-0B9B-A171-01FE-C51D234B86F7'}
				commandFeedback : REFERENCE TO MC_PlanarFeedback;
		(* Target position [mm] for the movement. *)
		targetPosition : LREAL;
		(* Dynamic constraints for this movement. *)
 {attribute 'GUID' := '6C0A73A2-C983-14C5-9BC7-15048F604248'}
		 {attribute 'Namespace' := 'Tc3_Physics'}
				constraint : REFERENCE TO IPlcDynamicConstraint;
	END_VAR
END_METHOD


	(* Initiates a relative movement for the y component. *)
	METHOD MoveRelativeY
	VAR_INPUT
		(* The feedback object for the command. *)
 {attribute 'GUID' := '8FADE443-0B9B-A171-01FE-C51D234B86F7'}
				commandFeedback : REFERENCE TO MC_PlanarFeedback;
		(* Target position [mm] for the movement. *)
		targetPosition : LREAL;
		(* Dynamic constraints for this movement. *)
 {attribute 'GUID' := '6C0A73A2-C983-14C5-9BC7-15048F604248'}
		 {attribute 'Namespace' := 'Tc3_Physics'}
				constraint : REFERENCE TO IPlcDynamicConstraint;
	END_VAR
END_METHOD


	(* Initiates a relative movement for the c component. *)
	METHOD MoveRelativeC
	VAR_INPUT
		(* The feedback object for the command. *)
 {attribute 'GUID' := '8FADE443-0B9B-A171-01FE-C51D234B86F7'}
				commandFeedback : REFERENCE TO MC_PlanarFeedback;
		(* Target position [deg] for the movement. *)
		targetPosition : LREAL;
		(* Dynamic constraints for this movement. *)
 {attribute 'GUID' := '6C0A73A2-C983-14C5-9BC7-15048F604248'}
		 {attribute 'Namespace' := 'Tc3_Physics'}
				constraint : REFERENCE TO IPlcDynamicConstraint;
	END_VAR
END_METHOD


	(* Initiates a movement for the x component. *)
	METHOD MoveVelocityX
	VAR_INPUT
		(* The feedback object for the command. *)
 {attribute 'GUID' := '8FADE443-0B9B-A171-01FE-C51D234B86F7'}
				commandFeedback : REFERENCE TO MC_PlanarFeedback;
		(* Target velocity [mm/s] for the movement. *)
		targetVelocity : LREAL;
		(* Dynamic constraints for this movement. *)
 {attribute 'GUID' := '6C0A73A2-C983-14C5-9BC7-15048F604248'}
		 {attribute 'Namespace' := 'Tc3_Physics'}
				constraint : REFERENCE TO IPlcDynamicConstraint;
	END_VAR
END_METHOD


	(* Initiates a movement for the y component. *)
	METHOD MoveVelocityY
	VAR_INPUT
		(* The feedback object for the command. *)
 {attribute 'GUID' := '8FADE443-0B9B-A171-01FE-C51D234B86F7'}
				commandFeedback : REFERENCE TO MC_PlanarFeedback;
		(* Target velocity [mm/s] for the movement. *)
		targetVelocity : LREAL;
		(* Dynamic constraints for this movement. *)
 {attribute 'GUID' := '6C0A73A2-C983-14C5-9BC7-15048F604248'}
		 {attribute 'Namespace' := 'Tc3_Physics'}
				constraint : REFERENCE TO IPlcDynamicConstraint;
	END_VAR
END_METHOD


	(* Initiates a movement for the c component. *)
	METHOD MoveVelocityC
	VAR_INPUT
		(* The feedback object for the command. *)
 {attribute 'GUID' := '8FADE443-0B9B-A171-01FE-C51D234B86F7'}
				commandFeedback : REFERENCE TO MC_PlanarFeedback;
		(* Target velocity [deg/s] for the movement. *)
		targetVelocity : LREAL;
		(* Dynamic constraints for this movement. *)
 {attribute 'GUID' := '6C0A73A2-C983-14C5-9BC7-15048F604248'}
		 {attribute 'Namespace' := 'Tc3_Physics'}
				constraint : REFERENCE TO IPlcDynamicConstraint;
	END_VAR
END_METHOD


	(* Initiates a rotation to adopt the orientation of the current track. *)
	METHOD AdoptTrackOrientation
	VAR_INPUT
		(* The feedback object for the command. *)
 {attribute 'GUID' := '8FADE443-0B9B-A171-01FE-C51D234B86F7'}
				commandFeedback : REFERENCE TO MC_PlanarFeedback;
		(* Dynamic constraints for this movement. *)
 {attribute 'GUID' := '6C0A73A2-C983-14C5-9BC7-15048F604248'}
		 {attribute 'Namespace' := 'Tc3_Physics'}
				constraint : REFERENCE TO IPlcDynamicConstraint;
		(* Options for the rotation. *)
 {attribute 'GUID' := 'CD2F9911-3022-4AB6-AED2-36E00F18E2B6'}
				options : REFERENCE TO ST_AdoptTrackOrientationOptions;
	END_VAR
END_METHOD


	(* Initiates a halt. *)
	METHOD Halt
	VAR_INPUT
		(* The feedback object for the command. *)
 {attribute 'GUID' := '8FADE443-0B9B-A171-01FE-C51D234B86F7'}
				commandFeedback : REFERENCE TO MC_PlanarFeedback;
		(* Dynamic constraints for this movement. *)
 {attribute 'GUID' := '6C0A73A2-C983-14C5-9BC7-15048F604248'}
		 {attribute 'Namespace' := 'Tc3_Physics'}
				constraint : REFERENCE TO IPlcDynamicConstraint;
	END_VAR
END_METHOD


	(* Starts enabling the Planar Mover. *)
	METHOD Enable
	VAR_INPUT
		(* The feedback object for the command. *)
 {attribute 'GUID' := '8FADE443-0B9B-A171-01FE-C51D234B86F7'}
				commandFeedback : REFERENCE TO MC_PlanarFeedback;
	END_VAR
END_METHOD


	(* Starts disabling the Planar Mover. *)
	METHOD Disable
	VAR_INPUT
		(* The feedback object for the command. *)
 {attribute 'GUID' := '8FADE443-0B9B-A171-01FE-C51D234B86F7'}
				commandFeedback : REFERENCE TO MC_PlanarFeedback;
	END_VAR
END_METHOD


	(* Starts resetting the Planar Mover. *)
	METHOD Reset
	VAR_INPUT
		(* The feedback object for the command. *)
 {attribute 'GUID' := '8FADE443-0B9B-A171-01FE-C51D234B86F7'}
				commandFeedback : REFERENCE TO MC_PlanarFeedback;
	END_VAR
END_METHOD


	(* Synchronizes the object state. Call once per PLC cycle. *)
	METHOD Update
END_METHOD


	(* Sets the position of the Planar Mover. Only possible if the Planar Mover is disabled. *)
	METHOD SetPosition
	VAR_INPUT
		(* The feedback object for the command. *)
 {attribute 'GUID' := '8FADE443-0B9B-A171-01FE-C51D234B86F7'}
				commandFeedback : REFERENCE TO MC_PlanarFeedback;
	END_VAR
	VAR_IN_OUT
		(* New position of the Planar Mover. *)
 {attribute 'GUID' := '12927DD4-F3D1-1B21-A804-08BCF50529B3'}
		 {attribute 'Namespace' := 'Tc3_Physics'}
				position : PositionXYC;
	END_VAR
END_METHOD


	(* Starts the external setpoint generation, the user must supply setpoints from this PLC cycle on in every PLC cycle. *)
	METHOD StartExternalSetpointGeneration
	VAR_INPUT
		(* The feedback object for the command. *)
 {attribute 'GUID' := '8FADE443-0B9B-A171-01FE-C51D234B86F7'}
				commandFeedback : REFERENCE TO MC_PlanarFeedback;
		(* Options for the movement. *)
 {attribute 'GUID' := '4CE91F7A-02E8-44B7-AB0B-38A598B51531'}
				options : REFERENCE TO ST_ExternalSetpointGenerationOptions;
	END_VAR
END_METHOD


	(* Ends the external setpoint generation, called after last SetExternalSetpoint (in the same PLC cycle). *)
	METHOD StopExternalSetpointGeneration
	VAR_INPUT
		(* The feedback object for the command. *)
 {attribute 'GUID' := '8FADE443-0B9B-A171-01FE-C51D234B86F7'}
				commandFeedback : REFERENCE TO MC_PlanarFeedback;
	END_VAR
END_METHOD


	(* Sets the external setpoint for the Planar Mover without reference system id (relative mode). Call once per PLC cycle during external setpoint generation. *)
	METHOD SetExternalSetpoint
	VAR_INPUT
		(* Position that is sent to the Planar Mover. *)
 {attribute 'GUID' := '5AC0538E-BDFA-4B58-A6B5-99E997DABADA'}
		 {attribute 'Namespace' := 'MC'}
				setPosition : MoverVector;
		(* Velocity that is sent to the Planar Mover. *)
 {attribute 'GUID' := '5AC0538E-BDFA-4B58-A6B5-99E997DABADA'}
		 {attribute 'Namespace' := 'MC'}
				setVelocity : MoverVector;
		(* Acceleration that is sent to the Planar Mover. *)
 {attribute 'GUID' := '5AC0538E-BDFA-4B58-A6B5-99E997DABADA'}
		 {attribute 'Namespace' := 'MC'}
				setAcceleration : MoverVector;
	END_VAR
END_METHOD


	(* Sets the external setpoint for the Planar Mover with corresponding reference system id. Call once per PLC cycle during external setpoint generation. *)
	METHOD SetExternalSetpointReferenceId
	VAR_INPUT
		(* The feedback object for the command. *)
 {attribute 'GUID' := '8FADE443-0B9B-A171-01FE-C51D234B86F7'}
				commandFeedback : REFERENCE TO MC_PlanarFeedback;
		(* Position that is sent to the Planar Mover. *)
 {attribute 'GUID' := '5AC0538E-BDFA-4B58-A6B5-99E997DABADA'}
		 {attribute 'Namespace' := 'MC'}
				setPosition : MoverVector;
		(* Velocity that is sent to the Planar Mover. *)
 {attribute 'GUID' := '5AC0538E-BDFA-4B58-A6B5-99E997DABADA'}
		 {attribute 'Namespace' := 'MC'}
				setVelocity : MoverVector;
		(* Acceleration that is sent to the Planar Mover. *)
 {attribute 'GUID' := '5AC0538E-BDFA-4B58-A6B5-99E997DABADA'}
		 {attribute 'Namespace' := 'MC'}
				setAcceleration : MoverVector;
		(* Part or coordinate system id. *)
 {attribute 'GUID' := '18071995-0000-0000-0000-00000000000F'}
				referenceSystemOid : OTCID;
	END_VAR
END_METHOD


	(* Raises a Planar Mover error, changing the Planar Mover state to ErrorPending (and then Error). *)
	{attribute 'hide'}
	METHOD RaiseError
	VAR_INPUT
		(* The feedback object for the command. *)
 {attribute 'GUID' := '8FADE443-0B9B-A171-01FE-C51D234B86F7'}
				commandFeedback : REFERENCE TO MC_PlanarFeedback;
		(* ErrorId of the Planar Mover error. *)
		errorId : UDINT;
	END_VAR
END_METHOD


	(* Adds the Planar Mover to the given Planar Group. *)
	METHOD AddToGroup
	VAR_INPUT
		(* The feedback object for the command. *)
 {attribute 'GUID' := '8FADE443-0B9B-A171-01FE-C51D234B86F7'}
				commandFeedback : REFERENCE TO MC_PlanarFeedback;
	END_VAR
	VAR_IN_OUT
		(* The Planar Group that the Planar Mover joins. *)
 {attribute 'GUID' := '311812D6-6FBB-A2BC-1644-8B3C8413ECE6'}
				group : MC_PlanarGroup;
	END_VAR
END_METHOD


	(* Removes the Planar Mover from its current Planar Group, i.e. disables collision checks. *)
	METHOD RemoveFromGroup
	VAR_INPUT
		(* The feedback object for the command. *)
 {attribute 'GUID' := '8FADE443-0B9B-A171-01FE-C51D234B86F7'}
				commandFeedback : REFERENCE TO MC_PlanarFeedback;
	END_VAR
END_METHOD


	(* Sets the values of the given position to the movers position values on the current part. *)
	METHOD GetPositionOnCurrentPart
	VAR_IN_OUT
		(* The position on the planar part. *)
 {attribute 'GUID' := '12927DD4-F3D1-1B21-A804-08BCF50529B3'}
		 {attribute 'Namespace' := 'Tc3_Physics'}
				position : PositionXYC;
	END_VAR
END_METHOD


	(* Gets the planned track trail for the mover's current track movement. *)
	METHOD GetTrackTrailInformation
	VAR_IN_OUT
		(* Track trail determining along which tracks the mover will move with the current movement on track. *)
 {attribute 'GUID' := 'F8359FE7-9712-A2F1-01A5-A9544A0C00B7'}
				trackTrail : MC_PlanarTrackTrail;
	END_VAR
END_METHOD


	(* Returns mover object info (type: mover, id: OID of nc mover). *)
	METHOD GetPlanarObjectInfo : PlanarObjectInfo
END_METHOD


{attribute 'monitoring' := 'call'}
	PROPERTY MoverHardwareOid : OTCID
GET
END_GET
END_PROPERTY

END_FUNCTION_BLOCK

// POUs/MC_PlanarFeedbackGearInPosOnTrack

	{attribute 'c++_compatible'}
	{attribute 'external_name' := 'MC_PlanarFeedbackGearInPosOnTrack_GUID_19C4A159_B3DC_ABFB_0783_72302E623B59'}
	{attribute 'TcIecLibraryType'}
	{attribute 'no_assign_warning'}
	(* Displays specific command status information for an associated GearInPosOnTrack command, given back by the MC Project. *)
	FUNCTION_BLOCK MC_PlanarFeedbackGearInPosOnTrack EXTENDS MC_PlanarFeedbackInSync


	(* Internal method *)
	{attribute 'hide'}
	METHOD FB_init : BOOL
	VAR_INPUT
		(*  if TRUE, the retain variables are initialized (warm start / cold start) *)
		bInitRetains : BOOL;
		(*  if TRUE, the instance afterwards gets moved into the copy code (online change) *)
		bInCopyCode : BOOL;
	END_VAR
END_METHOD


	(* Internal method *)
	{attribute 'hide'}
	METHOD FB_reinit : BOOL
END_METHOD


	(* Internal method *)
	{attribute 'hide'}
	METHOD FB_exit : BOOL
	VAR_INPUT
		(*  if TRUE, the exit method is called for exiting an instance that is copied afterwards (online change). *)
		bInCopyCode : BOOL;
	END_VAR
END_METHOD


	(* Updates internal state of the object. *)
	METHOD Update
END_METHOD

END_FUNCTION_BLOCK

// POUs/MC_PlanarFeedbackInSync

	{attribute 'c++_compatible'}
	{attribute 'external_name' := 'MC_PlanarFeedbackInSync_GUID_50AC999C_6346_A3A9_1181_475F95630E2B'}
	{attribute 'TcIecLibraryType'}
	{attribute 'no_explicit_call' :='do not call this POU directly'}
	{attribute 'no_assign_warning'}
	{attribute 'hide'}
	(* Base class for all specialized feedbacks featuring an inSync output. *)
	FUNCTION_BLOCK MC_PlanarFeedbackInSync EXTENDS MC_PlanarFeedbackBase 
	VAR_OUTPUT
		(* Indicates whether the mover is currently in sync with the master (within tolerance specified in the command options). *)
		inSync : BOOL;
	END_VAR
	VAR
		 {attribute 'hide'}
		_reserved1_1 : UINT_24_56;
	END_VAR


	(* Internal method *)
	{attribute 'hide'}
	METHOD FB_init : BOOL
	VAR_INPUT
		(*  if TRUE, the retain variables are initialized (warm start / cold start) *)
		bInitRetains : BOOL;
		(*  if TRUE, the instance afterwards gets moved into the copy code (online change) *)
		bInCopyCode : BOOL;
	END_VAR
END_METHOD


	(* Internal method *)
	{attribute 'hide'}
	METHOD FB_reinit : BOOL
END_METHOD


	(* Internal method *)
	{attribute 'hide'}
	METHOD FB_exit : BOOL
	VAR_INPUT
		(*  if TRUE, the exit method is called for exiting an instance that is copied afterwards (online change). *)
		bInCopyCode : BOOL;
	END_VAR
END_METHOD

END_FUNCTION_BLOCK

// POUs/MC_PlanarFeedbackGearInPosOnTrackWithMasterMover

	{attribute 'c++_compatible'}
	{attribute 'external_name' := 'MC_PlanarFeedbackGearInPosOnTrackWithMasterMover_GUID_A3111726_B59C_A154_0494_25C5C4FF630E'}
	{attribute 'TcIecLibraryType'}
	{attribute 'no_assign_warning'}
	(* Displays specific command status information for an associated GearInPosOnTrack command, given back by the MC Project. *)
	FUNCTION_BLOCK MC_PlanarFeedbackGearInPosOnTrackWithMasterMover EXTENDS MC_PlanarFeedbackInSync


	(* Internal method *)
	{attribute 'hide'}
	METHOD FB_init : BOOL
	VAR_INPUT
		(*  if TRUE, the retain variables are initialized (warm start / cold start) *)
		bInitRetains : BOOL;
		(*  if TRUE, the instance afterwards gets moved into the copy code (online change) *)
		bInCopyCode : BOOL;
	END_VAR
END_METHOD


	(* Internal method *)
	{attribute 'hide'}
	METHOD FB_reinit : BOOL
END_METHOD


	(* Internal method *)
	{attribute 'hide'}
	METHOD FB_exit : BOOL
	VAR_INPUT
		(*  if TRUE, the exit method is called for exiting an instance that is copied afterwards (online change). *)
		bInCopyCode : BOOL;
	END_VAR
END_METHOD


	(* Updates internal state of the object. *)
	METHOD Update
END_METHOD

END_FUNCTION_BLOCK
